// TwinCAT 3 PLC project AstroBROT
// Title: AstroBROT
// Company: BROT
// ProjectVersion: 0.4.5
// ProgramVersion: 3.1.4026.11
// libraries:
//   Tc2_Math, * (Beckhoff Automation GmbH)
//   Tc2_Standard, * (Beckhoff Automation GmbH)
//   Tc2_System, * (Beckhoff Automation GmbH)
//   Tc2_Utilities, * (Beckhoff Automation GmbH)
//   Tc3_Module, * (Beckhoff Automation GmbH)
// project tree:
//   POUs/FUNCTIONS/ ATAN2.TcPOU, CO_REFRACT_FORWARD.TcPOU, CT2LST.TcPOU, DateTime2JD.TcPOU, JD2LST.TcPOU, JD2JEPOCH.TcPOU, JD2OBLIQUITY.TcPOU, LMST2LAST.TcPOU, TEN.TcPOU
//   POUs/FUNCTION_BLOCKS/ FB_ALTAZ2HADEC.TcPOU, FB_CO_ABERRATION.TcPOU, FB_CO_REFRACT.TcPOU, FB_CO_NUTATE.TcPOU, FB_EQ2HOR.TcPOU, FB_HADEC2RADEC.TcPOU, FB_HADEC2ALTAZ.TcPOU, FB_HOR2EQ.TcPOU, FB_IAU2000B.TcPOU, FB_PRECESS.TcPOU, FB_RADEC2HADEC.TcPOU, FB_SUNPOS.TcPOU
//   GVLs/ Global_Version.TcGVL

// ---- GVLs/Global_Version.TcGVL
{attribute 'qualified_only'}
VAR_GLOBAL CONSTANT
	// Mirrors Beckhoff's own Global_Version.stLibVersion_* pattern (see ST_LibVersion),
	// which only covers Tc2_*/Tc3_* library references, not custom ones -- until now: this
	// GVL uses Beckhoff's own naming exactly, so it merges into a consumer's Global_Version.
	// Kept in sync with <ProjectVersion> in AstroBROT.plcproj at release time.
	stLibVersion_AstroBROT : ST_LibVersion := (
		iMajor := 0,
		iMinor := 4,
		iBuild := 5,
		iRevision := 0,
		nFlags := 1,
		sVersion := '0.4.5'
	);
END_VAR

// ---- POUs/FUNCTIONS/ATAN2.TcPOU
FUNCTION ATAN2 : LREAL
VAR_INPUT
	y		: LREAL;
	x		: LREAL;
END_VAR
VAR
END_VAR

(* source: https://de.wikipedia.org/wiki/Arctan2 *)
ATAN2 := 0.0;

IF x > 0 THEN
	ATAN2 := ATAN(y/x);
ELSIF x < 0 AND y > 0 THEN
	ATAN2 := ATAN(y/x) + PI;
ELSIF x < 0 AND y = 0 THEN
	ATAN2 := PI;
ELSIF x < 0 AND y < 0 THEN
	ATAN2 := ATAN(y/x) - PI;
ELSIF x = 0 AND y > 0 THEN
	ATAN2 := PI/2.0;
ELSIF x = 0 AND y < 0 THEN
	ATAN2 := -PI/2.0;
END_IF

END_FUNCTION

// ---- POUs/FUNCTIONS/CO_REFRACT_FORWARD.TcPOU
FUNCTION CO_REFRACT_FORWARD : LREAL
VAR_INPUT
	a			: LREAL; 			// The observed (apparent) altitude, in DEGREES.
	P			: LREAL := 1010.0;	// Pressure [in millibars]. Default is 1010 millibars.
	T			: LREAL := 0.0;		// Ground Temp [in Celsius].  Default is 0 Celsius.
END_VAR
VAR_OUTPUT
	clamped		: BOOL;				// TRUE if a, P or T was outside its valid range and has been limited
END_VAR
VAR
	ref			: LREAL;
	ref_lo		: LREAL;
	ref_hi		: LREAL;
	w			: LREAL;
	tk, gamma, beta, tan_z	: LREAL;
END_VAR
VAR CONSTANT
	d2r 		: LREAL := PI/180.0;
	// (n-1) * T / P for dry air at 0.55 um (IAG 1999 optical refractivity, as in eraRefco)
	k_gamma		: LREAL := 7.902649953145277E-5;
	// The two branches are blended linearly between these altitudes [DEGREES], so there is no step
	a_blend_lo	: LREAL := 14.0;
	a_blend_hi	: LREAL := 16.0;
END_VAR

(*Atmospheric refraction in DEGREES for an OBSERVED altitude a, pressure P [mbar] and temperature T [degC].
Dry air, 0.55 um, no humidity or wavelength input.

Below a_blend_lo (about 14 deg): the rational formula of the Explanatory Supplement to the Astronomical
Almanac, 2013, p.280 (eq. 7.91, not checked against the book).
From a_blend_hi (about 16 deg): dZ = A tan Z + B tan^3 Z with A and B from Green, Spherical Astronomy, 1987,
eq. 4.31 and beta from Stone (1996), exactly as ERFA's eraRefco (dry, wl = 0.55 um). eraRefco is
Copyright (C) 2013-2023 NumFOCUS Foundation, derived from SOFA, see NOTICE-erfa.md. Its documentation gives
62 mas worst case against ray tracing for zenith distances 15 to 75 deg (optical, humid air included).
Between the two: linear blend, so the result is continuous.

Accuracy of this implementation against an independent ray trace (testing/check_refraction_model.py, P 900 to
1013 mbar, T -15 to 30 degC): within 0.7 arcsec from 15 deg up, within 1.9 arcsec from 10 to 15 deg. NOT verified
below 10 deg, where the error reaches about 6 arcsec at 5 deg; do not rely on it near the horizon.

a, P and T are limited to [0, 90], [600, 1200] and [-40, 40] and clamped is set, so a caller can tell. A
below-horizon altitude therefore gets the horizon refraction.*)

clamped := (a < 0.0) OR (a > 90.0) OR (P < 600.0) OR (P > 1200.0) OR (T < -40.0) OR (T > 40.0);
a := LIMIT(0.0, a, 90.0);
P := LIMIT(600.0, P, 1200.0);
T := LIMIT(-40.0, T, 40.0);

IF a < a_blend_hi THEN
	ref_lo := P/(T+273.0)* (0.1594 + 0.0196 * a + 0.00002 * EXPT(a, 2)) / (1.0 + 0.505 * a + 0.0845 * EXPT(a, 2));
END_IF

IF a > a_blend_lo THEN
	tk := T + 273.15;
	gamma := k_gamma * P / tk;
	beta := 4.4474E-6 * tk;
	tan_z := TAN((90.0 - a) * d2r);
	ref_hi := (gamma * (1.0 - beta) * tan_z - gamma * (beta - gamma / 2.0) * tan_z * tan_z * tan_z) / d2r;
END_IF

IF a <= a_blend_lo THEN
	ref := ref_lo;
ELSIF a >= a_blend_hi THEN
	ref := ref_hi;
ELSE
	w := (a - a_blend_lo) / (a_blend_hi - a_blend_lo);
	ref := (1.0 - w) * ref_lo + w * ref_hi;
END_IF
CO_REFRACT_FORWARD :=  ref;

END_FUNCTION

// ---- POUs/FUNCTIONS/CT2LST.TcPOU
FUNCTION CT2LST : LREAL
VAR_INPUT
	lng: LREAL; // The longitude in degrees (east of Greenwich) of the place for which the local sidereal time is desired, scalar.   The Greenwich mean sidereal time (GMST) can be found by setting Lng = 0.
	jd:	LREAL; // this is the Julian date of time in question
END_VAR
VAR
	t0,t,theta: LREAL;
END_VAR
VAR CONSTANT
	jd2000: LREAL := 2451545.0;
END_VAR

(* https://github.com/wlandsman/IDLAstro/blob/master/pro/ct2lst.pro 

;+
; NAME:
;     CT2LST
; PURPOSE:
;     To convert from Local Civil Time to Local Mean Sidereal Time.
;
; CALLING SEQUENCE:
;     CT2LST, Lst, Lng, Tz, Time, [Day, Mon, Year] 
;                       or
;     CT2LST, Lst, Lng, dummy, JD
;
; INPUTS:
;     Lng  - The longitude in degrees (east of Greenwich) of the place for 
;            which the local sidereal time is desired, scalar.   The Greenwich 
;            mean sidereal time (GMST) can be found by setting Lng = 0.
;     Tz  - The time zone of the site in hours, positive East  of the Greenwich
;           meridian (ahead of GMT).  Use this parameter to easily account 
;           for Daylight Savings time (e.g. -4=EDT, -5 = EST/CDT), scalar
;           This parameter is not needed (and ignored) if Julian date is 
;           supplied.    ***Note that the sign of TZ was changed in July 2008
;           to match the standard definition.*** 
;     Time or JD  - If more than four parameters are specified, then this is 
;               the time of day of the specified date in decimal hours.  If 
;               exactly four parameters are specified, then this is the 
;               Julian date of time in question, scalar or vector
;
; OPTIONAL INPUTS:
;      Day -  The day of the month (1-31),integer scalar or vector
;      Mon -  The month, in numerical format (1-12), integer scalar or vector
;      Year - The 4 digit year (e.g. 2008), integer scalar or vector
;
; OUTPUTS:
;       Lst   The Local Sidereal Time for the date/time specified in hours.
;
; RESTRICTIONS:
;       If specified, the date should be in numerical form.  The year should
;       appear as yyyy.
;
; PROCEDURE:
;       The Julian date of the day and time is question is used to determine
;       the number of days to have passed since 0 Jan 2000.  This is used
;       in conjunction with the GST of that date to extrapolate to the current
;       GST; this is then used to get the LST.    See Astronomical Algorithms
;       by Jean Meeus, p. 84 (Eq. 11-4) for the constants used.
;
; EXAMPLE:
;       Find the Greenwich mean sidereal time (GMST) on 2008 Jul 30 at 15:53 pm
;       in Baltimore, Maryland (longitude=-76.72 degrees).   The timezone is 
;       EDT or tz=-4
;
;       IDL> CT2LST, lst, -76.72, -4,ten(15,53), 30, 07, 2008
;
;               ==> lst =  11.356505  hours  (= 11h 21m 23.418s)
;
;       The Web site  http://tycho.usno.navy.mil/sidereal.html contains more
;       info on sidereal time, as well as an interactive calculator.
; PROCEDURES USED:
;       jdcnv - Convert from year, month, day, hour to julian date
;
; MODIFICATION HISTORY:
;     Adapted from the FORTRAN program GETSD by Michael R. Greason, STX, 
;               27 October 1988.
;     Use IAU 1984 constants Wayne Landsman, HSTX, April 1995, results 
;               differ by about 0.1 seconds  
;     Longitudes measured *east* of Greenwich   W. Landsman    December 1998
;     Time zone now measure positive East of Greenwich W. Landsman July 2008
;     Remove debugging print statement  W. Landsman April 2009
;-

*)

t0 := jd - jd2000;
t := t0/36525.0;
// Compute GST in seconds.
theta := 280.46061837 + (360.98564736629 * t0) + EXPT(t, 2)*(0.000387933 - (t/ 3871.0E4));
//theta := 100.46061837 + 36000.770053608*t0 + 0.000387933*EXPT(t0,2) - EXPT(t0,3)/3871000.0;
// Compute LST in hours.
CT2LST := ( theta + lng)/15.0;
CT2LST := MODABS(CT2LST, 24.0);

END_FUNCTION

// ---- POUs/FUNCTIONS/DateTime2JD.TcPOU
FUNCTION DateTime2JD : LREAL
VAR_INPUT
	epoch			: TIMESTRUCT;
END_VAR
VAR
	a, y, m, jdn	: LREAL;
END_VAR

// Julian Date of a TIMESTRUCT (Meeus, Astronomical Algorithms, ch. 7; integer-day formula of the Gregorian calendar).
//
// - epoch must be UTC. The function does not convert or check the time zone; a local time gives a JD that is off by the
//   UTC offset, and with it the sidereal time (15 degrees per hour).
// - Gregorian calendar only, i.e. valid from 1582-10-15. Earlier dates would need the Julian-calendar formula.
// - No validation. Out-of-range fields roll over (month 13 is January of the next year, 30 February is 2 March), and an
//   all-zero TIMESTRUCT (e.g. a clock that has not been synchronised yet) gives 1721027.5, which is not a usable time.
a := FLOOR((14.0 - epoch.wMonth)/12.0);
y := epoch.wYear + 4800.0 - a;
m := epoch.wMonth + 12.0*a - 3.0;

jdn := epoch.wDay + FLOOR((153*m + 2)/5) + 365.0*y + FLOOR(y/4) - FLOOR(y/100) + FLOOR(y/400) - 32045.0;

DateTime2JD := jdn
			+ (epoch.wHour-12.0)/24.0
			+ (epoch.wMinute/1440.0) 
			+ (epoch.wSecond/86400.0)
			+ (DWORD_TO_REAL(epoch.wMilliseconds)/86400000.0);

END_FUNCTION

// ---- POUs/FUNCTIONS/JD2LST.TcPOU
FUNCTION JD2LST : LREAL
VAR_INPUT
	jd			: LREAL;	// Julian date, UTC time scale
	lon			: LREAL;	// longitude in degrees
	dut1		: LREAL := 0.0;	// UT1-UTC in seconds (IERS, |dut1| < 0.9), 0 treats UTC as UT1
END_VAR
VAR
	ut1			: LREAL;
	T			: LREAL;
	theta0		: LREAL;
END_VAR
VAR CONSTANT
	jd2000		: LREAL := 2451545.0;
END_VAR

// following https://squarewidget.com/astronomical-calculations-sidereal-time/
ut1 := jd + dut1 / 86400.0;
T := ((ut1 - jd2000) / 36525.0);
theta0 := 280.46061837 + 360.98564736629 * (ut1 - jd2000) + (0.000387933 * T * T) - (T * T * T / 38710000.0); // (12.4)

// LST is only defined from 0 to 360
JD2LST := MODABS(theta0 + lon, 360.0); // LST in degrees

END_FUNCTION

// ---- POUs/FUNCTIONS/JD2JEPOCH.TcPOU
FUNCTION JD2JEPOCH : LREAL
VAR_INPUT
	jd			: LREAL;	// Julian date
END_VAR
VAR CONSTANT
	jd2000		: LREAL := 2451545.0;
END_VAR

// Julian epoch (equinox) of jd, e.g. for precession
JD2JEPOCH := (jd - jd2000)/365.25 + 2000.0;

END_FUNCTION

// ---- POUs/FUNCTIONS/JD2OBLIQUITY.TcPOU
FUNCTION JD2OBLIQUITY : LREAL
VAR_INPUT
	jd			: LREAL;	// Julian date
	d_eps		: LREAL;	// nutation in obliquity in arcsec (FB_IAU2000B)
END_VAR
VAR
	T			: LREAL;
	eps0		: LREAL;
END_VAR
VAR CONSTANT
	d2r			: LREAL := PI/180.0;
	jd2000		: LREAL := 2451545.0;
END_VAR

// Julian centuries from J2000 of jd
T := (jd - jd2000)/36525.0;

// mean obliquity of the ecliptic in arcsec
eps0 := 23.4392911*3600.0 - 46.8150*T - 0.00059*EXPT(T, 2) + 0.001813*EXPT(T, 3);

// TRUE obliquity of the ecliptic in radians
JD2OBLIQUITY := (eps0 + d_eps)/3600.0*d2r;

END_FUNCTION

// ---- POUs/FUNCTIONS/LMST2LAST.TcPOU
FUNCTION LMST2LAST : LREAL
VAR_INPUT
	lmst		: LREAL;	// local mean sidereal time in degrees
	d_psi		: LREAL;	// nutation in longitude in arcsec (FB_IAU2000B)
	eps			: LREAL;	// TRUE obliquity of the ecliptic in radians (JD2OBLIQUITY)
END_VAR

// local APPARENT sidereal time in degrees: add the equation of the equinoxes
LMST2LAST := lmst + d_psi*COS(eps)/3600.0;

END_FUNCTION

// ---- POUs/FUNCTIONS/TEN.TcPOU
FUNCTION TEN : LREAL
VAR_INPUT
	dd, mm, ss	: LREAL;
END_VAR
VAR
	fSign	: LREAL;
END_VAR

// as IDLAstro's ten: a minus sign on any element makes the whole value negative, so TEN(-5, 30, 0) = -5.5
// (unlike IDL, a literal -0.0 is not recognised as negative)
IF (dd < 0.0) OR (mm < 0.0) OR (ss < 0.0) THEN
	fSign := -1.0;
ELSE
	fSign := 1.0;
END_IF
TEN := fSign * (ABS(dd) + (ABS(mm)/60.0) + (ABS(ss)/3600.0));

END_FUNCTION

// ---- POUs/FUNCTION_BLOCKS/FB_ALTAZ2HADEC.TcPOU
FUNCTION_BLOCK FB_ALTAZ2HADEC
VAR_INPUT
	alt			: LREAL;	// the local apparent altitude, in DEGREES
	az			: LREAL;	// the local apparent azimuth, in DEGREES
	lat			: LREAL;	// the local geodetic latitude, in DEGREES
END_VAR
VAR_OUTPUT
	ha			: LREAL;	// the local apparent hour angle, in DEGREES
	dec			: LREAL;	// the local apparent declination, in DEGREES
END_VAR
VAR
	alt_r		: LREAL;
	az_r		: LREAL;
	lat_r		: LREAL;
	sindec		: LREAL;
END_VAR
VAR CONSTANT
	d2r			: LREAL := PI/180.0;
	r2d			: LREAL := 180.0/PI;
	//h2r:	LREAL := PI/12.0;
	//h2d:	LREAL := 15.0;
END_VAR

(*https://github.com/wlandsman/IDLAstro/blob/master/pro/

  NAME:
    ALTAZ2HADEC
 PURPOSE:
    Convert Horizon (Alt-Az) coordinates to Hour Angle and Declination.
 EXPLANATION::
    Can deal with the NCP singularity.    Intended mainly to be used by
    program hor2eq.pro
 CALLING SEQUENCE:
   ALTAZ2HADEC, alt, az, lat, ha, dec

 INPUTS
   alt - the local apparent altitude, in DEGREES, scalar or vector
   az  - the local apparent azimuth, in DEGREES, scalar or vector,
         measured EAST of NORTH!!!  If you have measured azimuth west-of-south
        (like the book MEEUS does), convert it to east of north via:
                       az = (az + 180) mod 360

   lat -  the local geodetic latitude, in DEGREES, scalar or vector.

 OUTPUTS
   ha  -  the local apparent hour angle, in DEGREES.  The hour angle is the 
          time that right ascension of 0 hours crosses the local meridian.  
          It is unambiguously defined.
   dec -  the local apparent declination, in DEGREES.

 EXAMPLE:
     Arcturus is observed at an apparent altitude of 59d,05m,10s and an 
     azimuth (measured east of north) of 133d,18m,29s while at the 
     latitude of +43.07833 degrees.
     What are the local hour angle and declination of this object?

     IDL> altaz2hadec, ten(59,05,10), ten(133,18,29), 43.07833, ha, dec
     ===> Hour angle ha = 336.683 degrees
          Declination, dec = 19.1824 degrees

       The widely available XEPHEM code gets:
                 Hour Angle = 336.683
                 Declination = 19.1824

 REVISION HISTORY:
    Written  Chris O'Dell Univ. of Wisconsin-Madison May 2002*)

alt_r  := alt*d2r;
az_r := az*d2r;
lat_r := lat*d2r;

//******************************************************************************
// find local HOUR ANGLE (in degrees, from 0. to 360.)
ha := atan2( (-SIN(az_r)*COS(alt_r)), (-COS(az_r)*SIN(lat_r)*COS(alt_r)+SIN(alt_r)*COS(lat_r)));
ha := ha / d2r;
IF ha < 0.0 THEN 
	ha := ha + 360.0;
END_IF
ha := MODABS(ha, 360.0);

// Find declination (positive if north of Celestial Equator, negative if south)
sindec := SIN(lat_r)*SIN(alt_r) + COS(lat_r)*COS(alt_r)*COS(az_r);
// convert dec to degrees
dec := ASIN(LIMIT(-1.0, sindec, 1.0))/d2r;   // clamp: at the celestial pole rounding gives 1 + 2.2E-16, and ASIN of that is NaN

END_FUNCTION_BLOCK

// ---- POUs/FUNCTION_BLOCKS/FB_CO_ABERRATION.TcPOU
FUNCTION_BLOCK FB_CO_ABERRATION
VAR_INPUT
	jd			: LREAL;		// Julian Date
	ra			: LREAL;		// RA in degrees
	dec			: LREAL; 		// Dec in degrees
	eps 		: LREAL := 0.0;
END_VAR
VAR_OUTPUT
	d_ra		: LREAL;
	d_dec		: LREAL;
END_VAR
VAR
	sunpos		: FB_SUNPOS;
	nutate		: FB_IAU2000B;
	sunra		: LREAL;
	sundec		: LREAL;
	sunlon		: LREAL;
	d_psi		: LREAL;
	d_epsilon	: LREAL; 
	eps_loc		: LREAL;		// obliquity in radians, eps or calculated if eps = 0
	t, e, peri, cd, sd, ce, te, cp, sp, cs, ss, ca, sa, term1, term2, term3, term4: LREAL;
END_VAR
VAR CONSTANT
	d2r 		: LREAL := PI/180.0;
	k			: LREAL := 20.49552; 	//constant of aberration, in arcseconds
	
END_VAR

(* https://github.com/wlandsman/IDLAstro/blob/master/pro/co_aberration.pro
;+
;  NAME:
;     CO_ABERRATION
; PURPOSE:
;     Calculate changes to Ra and Dec due to the effect of annual aberration 
; EXPLANATION:
;      as described in Meeus, Chap 23.
; CALLING SEQUENCE:
;      co_aberration, jd, ra, dec, d_ra, d_dec, [EPS = ]
; INPUTS
;       jd      : Julian Date [scalar or vector]
;       ra, dec : ra  and dec's in degrees
;
; OUTPUTS
;       d_ra, d_dec: the corrections to ra and dec due to aberration in 
;                    degrees.  (These values can be added to the true RA 
;                    and dec to get the apparent position).   Note that d_ra
;                     is *not* multiplied by cos(dec), so that 
;                     apparent_ra = ra + d_ra. 
; OPTIONAL INPUT KEYWORD:
;       eps : set this to the true obliquity of the ecliptic (in radians), or
;         it will be set for you if you don't know it (in that case, set it to
;                 an empty variable).
; NOTES:
;  These formula are from Meeus, Chapters 23.  Accuracy is much better than 1 
;   arcsecond.
;
;   The maximum deviation due to annual aberration is 20.49" and occurs when the
;   Earth velocity is perpendicular to the direction of the star.
;
; REVISION HISTORY:
;   Written, June 2002,      Chris O'Dell, U. of Wisconsin
;   Fix error with vector input   W. Landsman   June 2009
;   June 2009 update fixed case where JD was scalar but RA,Dec were vectors, but 
;     broke the case when both JD and RA,Dec were vectors Aug 2012 W. Landsman
;   Further fix when JD is 1 element vector  W. Landsman
;
;	UPDATE: HAS BEEN REWORKED FOR THE COORD STRUCTURE -> OUTPUT IS IN DEGREES
*)

T := (jd -2451545.0)/36525.0; // julian centuries from J2000 of jd.

IF eps = 0.0 THEN
	// must calculate obliquity of ecliptic
	nutate(jd := jd,
		d_psi => d_psi, 
		d_eps => d_epsilon); //d_psi and d_epsilon in arcsec
	// TRUE obliquity OF the ecliptic in radians
	eps_loc := JD2OBLIQUITY(jd, d_epsilon);
ELSE
	eps_loc := eps;
END_IF

sunpos(jd := jd, ra => sunra, dec => sundec, longmed => sunlon);

// Earth's orbital eccentricity
e := 0.016708634 - 0.000042037*T - 0.0000001267*EXPT(T, 2);
// longitude of perihelion, in degrees 
peri := 102.93735 + 1.71946*T + 0.00046*EXPT(T, 2);

//Useful Trig Functions
cd := COS(dec*d2r);		sd := SIN(dec*d2r);
ce := COS(eps_loc); 	te := TAN(eps_loc);
cp := COS(peri*d2r);	sp := SIN(peri*d2r);
cs := COS(sunlon*d2r);	ss := SIN(sunlon*d2r);
ca := COS(ra*d2r);		sa := SIN(ra*d2r);

term1 := (ca*cs*ce + sa*ss)/cd;
term2 := (ca*cp*ce + sa*sp)/cd;
term3 := (cs*ce*(te*cd - sa*sd) + ca*sd*ss);
term4 := (cp*ce*(te*cd - sa*sd) + ca*sd*sp);

d_ra := (-k * term1 + e*k * term2)/3600;
d_dec := (-k * term3 + e*k * term4)/3600;

END_FUNCTION_BLOCK

// ---- POUs/FUNCTION_BLOCKS/FB_SUNPOS.TcPOU
FUNCTION_BLOCK FB_SUNPOS
VAR_INPUT
	jd				: LREAL;		// Julian Date
END_VAR
VAR_OUTPUT
	ra				: LREAL;		// right ascension
	dec				: LREAL;		// declination of the sun 
	longmed			: LREAL;		// longitude
	oblt			: LREAL;		// True Obliquity
END_VAR
VAR
	t				: LREAL;		//  Julian centuries FROM 1900.0
	l				: LREAL;		//  sun's mean longitude
	me				: LREAL;		// Earth's mean anomaly
	ellcor			: LREAL;		// ellipticity of the orbit
	mv				: LREAL;		// mean anomaly of Venus
	vencorr			: LREAL;		
	mm				: LREAL;		
	marscorr		: LREAL;		
	mj				: LREAL;		
	jupcorr			: LREAL;		
	d				: LREAL;		
	longterm		: LREAL;		
	mooncorr		: LREAL;		
	omega			: LREAL;
END_VAR
VAR CONSTANT
	d2r				: LREAL := PI/180.0; // Pi/180
END_VAR

(* https://github.com/wlandsman/IDLAstro/blob/master/pro/
NOTES:
;       Patrick Wallace (Rutherford Appleton Laboratory, UK) has tested the
;       accuracy of a C adaptation of the sunpos.pro code and found the 
;       following results.   From 1900-2100 SUNPOS  gave 7.3 arcsec maximum 
;       error, 2.6 arcsec RMS.  Over the shorter interval 1950-2050 the figures
;       were 6.4 arcsec max, 2.2 arcsec RMS.  
;
;       The returned ra and Dec are in the given date's equinox.
;
;       Procedure was extensively revised in May 1996, and the new calling
;       sequence is incompatible with the old one.source: https://idlastro.gsfc.nasa.gov/ftp/pro/astro/sunpos.pro *)

//  form TIME in Julian centuries FROM 1900.0
t := (jd - 2415020.0) / 36525.0;

//  form sun's mean longitude
l := (279.696678 + LMOD(36000.768925 * t, 360.0)) * 3600.0;

//  allow for ellipticity of the orbit (equation of centre) using the Earth's mean anomaly ME
me := 358.475844 + LMOD(35999.049750 * t, 360.0);
ellcor  := (6910.1 - 17.2 * t) * SIN(me * d2r) + 72.3 * SIN(2.0 * me*d2r);
l := l + ellcor;
 
// allow FOR the Venus perturbations using the mean anomaly OF Venus MV
mv := 212.603219 + LMOD(58517.803875 * t, 360.0);
vencorr := 4.8 * COS((299.1017 + mv - me)*d2r) + 
           5.5 * COS((148.3133 +  2.0 * mv  -  2.0 * me )*d2r) + 
           2.5 * COS((315.9433 +  2.0 * mv  -  3.0 * me )*d2r) + 
           1.6 * COS((345.2533 +  3.0 * mv  -  4.0 * me )*d2r) + 
           1.0 * COS((318.15   +  3.0 * mv  -  5.0 * me )*d2r);
l := l + vencorr;

//  Allow FOR the Mars perturbations using the mean anomaly OF Mars MM
mm := 319.529425  +  LMOD( 19139.858500 * t,  360.0 );
marscorr := 2.0 * COS((343.8883 -  2.0 * mm  +  2.0 * me)*d2r ) + 
            1.8 * COS((200.4017 -  2.0 * mm  + me) * d2r);
l := l + marscorr;

// Allow FOR the Jupiter perturbations using the mean anomaly OF Jupiter MJ
mj := 225.328328  +  LMOD( 3034.6920239 * t,  360.0 );
jupcorr := 7.2 * COS(( 179.5317 - mj + me )*d2r) + 
           2.6 * COS((263.2167  -  MJ ) *d2r) + 
           2.7 * COS(( 87.1450  -  2.0 * mj  +  2.0 * me ) *d2r) + 
           1.6 * COS((109.4933  -  2.0 * mj  +  me ) *d2r);
l := l + jupcorr;

// Allow FOR the Moons perturbations using the mean elongation OF the Moon from the Sun D
d := 350.7376814  + LMOD(445267.11422 * t,  360.0);
mooncorr  := 6.5 * SIN(d * d2r);
l := l + mooncorr;

// Allow for long period terms
longterm := 6.4 * SIN((231.19  +  20.20 * t) * d2r);
l :=  l + longterm;
l :=  LMOD(l + 2592000.0,  1296000.0); 
longmed := l / 3600.0;

// Allow for Aberration
l :=  l - 20.5;

// Allow for Nutation using the longitude of the Moons mean node OMEGA
omega := 259.183275 - LMOD(1934.142008 * t, 360.0);
l :=  l - 17.2 * SIN(omega * d2r);

// Form the True Obliquity
oblt := 23.452294 - 0.0130125 * t + (9.2 * COS(omega * d2r)) / 3600.0;

// Form Right Ascension AND Declination
l := l / 3600.0;
ra := ATAN2(SIN(l * d2r) * COS(oblt * d2r), COS(l * d2r));
dec := ASIN(SIN(l * d2r) * SIN(oblt * d2r));
 
ra := ra/d2r;
ra := MODABS(ra, 360.0);
dec := dec/d2r;

END_FUNCTION_BLOCK

// ---- POUs/FUNCTION_BLOCKS/FB_IAU2000B.TcPOU
FUNCTION_BLOCK FB_IAU2000B
VAR_INPUT
	jd: LREAL;
END_VAR
VAR_OUTPUT
	// unit: arcsec
	// d_psi and d_eps are not the pure IAU 2000B nutation: constant offsets standing in for the planetary terms
	// and the frame bias are added (-0.0433585 and -0.0084531 arcsec, see the end of the implementation)
	d_psi : LREAL := 0.0; 
	d_eps : LREAL := 0.0;
END_VAR
VAR
	t	: LREAL;
	m_l, m_l_, m_f, m_d, m_om : LREAL;
	theta, s_theta, c_theta : LREAL;
	d_p, d_e : LREAL := 0.0;
	i : INT;
END_VAR
VAR CONSTANT
	d2r				: LREAL := PI/180.0;
	asec2r			: LREAL := PI/(180*3600);
	asec360			: LREAL := 3600*360;
	jd2000			: LREAL := 2451545.0;
	// number of luni-solar terms of IAU 2000B
	n_terms			: INT := 77;
	// Luni-Solar argument multipliers:
	l	: ARRAY[1..77] OF LREAL := [0, 0, 0, 0, 0, 0, 1, 0, 1, 0, 0, -1, -1, 1, -1, -1, 1, -2, 0, 0, 0, -2, 2, 1, -1, 2, 0, 0, -1, 0, 0, 1, 0, -1, 0, 1, -2, 0, 0, 0, 0, 1, 2, -2, 2, 0, 0, -1, 2, 1, 0, 1, -2, 3, 0, 1, 0, -1, -1, 0, -2, 1, 2, -1, 1, 1, -1, 1, -1, 0, -1, -1, 0, 1, -2, -1, 1];
	l_	: ARRAY[1..77] OF LREAL := [0, 0, 0, 0, 1, 1, 0, 0, 0, -1, 0, 0, 0, 0, 0, 0, 0, 0, 0, 0, -2, 0, 0, 0, 0, 0, 0, 1, 0, 2, 0, 0, -1, 0, 2, 0, 0, 1, 0, -1, 0, 0, 0, 0, 0, -1, 0, -1, 0, 0, 1, -1, 0, 0, -1, -1, 0, -1, 0, -1, 0, 1, 0, 1, 1, 0, 0, 0, 0, 0, 0, 1, -2, 0, 0, 0, 1];
	f 	: ARRAY[1..77] OF LREAL := [0, 2, 2, 0, 0, 2, 0, 2, 2, 2, 2, 2, 0, 0, 0, 2, 2, 2, 0, 2, 2, 0, 2, 2, 2, 0, 2, 0, 0, 2, -2, 0, 0, 2, 0, 2, 2, 2, 2, 2, 0, 2, 2, 0, 2, 2, 0, 0, 0, 0, 2, 0, 2, 2, 0, 2, 0, 2, 2, 2, 0, 2, 0, 0, 0, 2, 2, 0, 0, 2, 2, 0, 2, 2, 2, 0, 2];
	d 	: ARRAY[1..77] OF LREAL := [0, -2, 0, 0, 0, -2, 0, 0, 0, -2, -2, 0, 2, 0, 0, 2, 0, 0, 2, 2, -2, 2, 0, -2, 0, 0, 0, 0, 2, -2, 2, -2, 0, 2, 0, 2, 0, 0, 2, 0, 2, -2, -2, 2, 0, -2, -2, 2, -2, 2, -2, 0, 0, 0, 2, 0, 1, 2, 0, 2, 0, 0, 0, 1, 0, 0, -2, 0, 1, 1, 4, 1, -2, 2, 2, 0, -2];
	om	: ARRAY[1..77] OF LREAL := [1, 2, 2, 2, 0, 2, 0, 1, 2, 2, 1, 2, 0, 1, 1, 2, 1, 1, 0, 2, 2, 0, 2, 2, 1, 0, 0, 1, 1, 2, 0, 1, 1, 1, 0, 2, 0, 2, 1, 2, 1, 1, 2, 1, 1, 1, 1, 0, 1, 0, 1, 0, 2, 2, 0, 2, 0, 2, 0, 2, 1, 2, 1, 0, 0, 0, 1, 2, 0, 2, 2, 1, 1, 1, 2, 2, 2];
	//  Luni-Solar nutation coefficients, unit 1e-7 arcsec:
	A 	: ARRAY[1..77] OF LREAL := [-172064161.0, -13170906.0, -2276413.0, 2074554.0, 1475877.0, -516821.0, 711159.0, -387298.0, -301461.0, 215829.0, 128227.0, 123457.0, 156994.0, 63110.0, -57976.0, -59641.0, -51613.0, 45893.0, 63384.0, -38571.0, 32481.0, -47722.0, -31046.0, 28593.0, 20441.0, 29243.0, 25887.0, -14053.0, 15164.0, -15794.0, 21783.0, -12873.0, -12654.0, -10204.0, 16707.0, -7691.0, -11024.0, 7566.0, -6637.0, -7141.0, -6302.0, 5800.0, 6443.0, -5774.0, -5350.0, -4752.0, -4940.0, 7350.0, 4065.0, 6579.0, 3579.0, 4725.0, -3075.0, -2904.0, 4348.0, -2878.0, -4230.0, -2819.0, -4056.0, -2647.0, -2294.0, 2481.0, 2179.0, 3276.0, -3389.0, 3339.0, -1987.0, -1981.0, 4026.0, 1660.0, -1521.0, 1314.0, -1283.0, -1331.0, 1383.0, 1405.0, 1290.0];
	A1 	: ARRAY[1..77] OF LREAL := [-174666.0, -1675.0, -234.0, 207.0, -3633.0, 1226.0, 73.0, -367.0, -36.0, -494.0, 137.0, 11.0, 10.0, 63.0, -63.0, -11.0, -42.0, 50.0, 11.0, -1.0, 0.0, 0.0, -1.0, 0.0, 21.0, 0.0, 0.0, -25.0, 10.0, 72.0, 0.0, -10.0, 11.0, 0.0, -85.0, 0.0, 0.0, -21.0, -11.0, 21.0, -11.0, 10.0, 0.0, -11.0, 0.0, -11.0, -11.0, 0.0, 0.0, 0.0, 0.0, 0.0, 0.0, 0.0, 0.0, 0.0, 0.0, 0.0, 0.0, 0.0, 0.0, 0.0, 0.0, 0.0, 0.0, 0.0, 0.0, 0.0, 0.0, 0.0, 0.0, 0.0, 0.0, 0.0, 0.0, 0.0, 0.0];
	A2 	: ARRAY[1..77] OF LREAL := [33386.0, -13696.0, 2796.0, -698.0, 11817.0, -524.0, -872.0, 380.0, 816.0, 111.0, 181.0, 19.0, -168.0, 27.0, -189.0, 149.0, 129.0, 31.0, -150.0, 158.0, 0.0, -18.0, 131.0, -1.0, 10.0, -74.0, -66.0, 79.0, 11.0, -16.0, 13.0, -37.0, 63.0, 25.0, -10.0, 44.0, -14.0, -11.0, 25.0, 8.0, 2.0, 2.0, -7.0, -15.0, 21.0, -3.0, -21.0, -8.0, 6.0, -24.0, 5.0, -6.0, -2.0, 15.0, -10.0, 8.0, 5.0, 7.0, 5.0, 11.0, -10.0, -7.0, -2.0, 1.0, 5.0, -13.0, -6.0, 0.0, -353.0, -5.0, 9.0, 0.0, 0.0, 8.0, -2.0, 4.0, 0.0];
	B 	: ARRAY[1..77] OF LREAL := [92052331.0, 5730336.0, 978459.0, -897492.0, 73871.0, 224386.0, -6750.0, 200728.0, 129025.0, -95929.0, -68982.0, -53311.0, -1235.0, -33228.0, 31429.0, 25543.0, 26366.0, -24236.0, -1220.0, 16452.0, -13870.0, 477.0, 13238.0, -12338.0, -10758.0, -609.0, -550.0, 8551.0, -8001.0, 6850.0, -167.0, 6953.0, 6415.0, 5222.0, 168.0, 3268.0, 104.0, -3250.0, 3353.0, 3070.0, 3272.0, -3045.0, -2768.0, 3041.0, 2695.0, 2719.0, 2720.0, -51.0, -2206.0, -199.0, -1900.0, -41.0, 1313.0, 1233.0, -81.0, 1232.0, -20.0, 1207.0, 40.0, 1129.0, 1266.0, -1062.0, -1129.0, -9.0, 35.0, -107.0, 1073.0, 854.0, -553.0, -710.0, 647.0, -700.0, 672.0, 663.0, -594.0, -610.0, -556.0];
	B1 	: ARRAY[1..77] OF LREAL := [9086.0, -3015.0, -485.0, 470.0, -184.0, -677.0, 0.0, 18.0, -63.0, 299.0, -9.0, 32.0, 0.0, 0.0, 0.0, -11.0, 0.0, -10.0, 0.0, -11.0, 0.0, 0.0, -11.0, 10.0, 0.0, 0.0, 0.0, -2.0, 0.0, -42.0, 0.0, 0.0, 0.0, 0.0, -1.0, 0.0, 0.0, 0.0, 0.0, 0.0, 0.0, 0.0, 0.0, 0.0, 0.0, 0.0, 0.0, 0.0, 0.0, 0.0, 0.0, 0.0, 0.0, 0.0, 0.0, 0.0, 0.0, 0.0, 0.0, 0.0, 0.0, 0.0, 0.0, 0.0, 0.0, 0.0, 0.0, 0.0, 0.0, 0.0, 0.0, 0.0, 0.0, 0.0, 0.0, 0.0, 0.0];
	B2	: ARRAY[1..77] OF LREAL := [15377.0, -4587.0, 1374.0, -291.0, -1924.0, -174.0, 358.0, 318.0, 367.0, 132.0, 39.0, -4.0, 82.0, -9.0, -75.0, 66.0, 78.0, 20.0, 29.0, 68.0, 0.0, -25.0, 59.0, -3.0, -3.0, 13.0, 11.0, -45.0, -1.0, -5.0, 13.0, -14.0, 26.0, 15.0, 10.0, 19.0, 2.0, -5.0, 14.0, 4.0, 4.0, -1.0, -4.0, -5.0, 12.0, -3.0, -9.0, 4.0, 1.0, 2.0, 1.0, 3.0, -1.0, 7.0, 2.0, 4.0, -2.0, 3.0, -2.0, 5.0, -4.0, -3.0, -2.0, 0.0, -2.0, 1.0, -2.0, 0.0, -139.0, -2.0, 4.0, 0.0, 0.0, 4.0, -2.0, 2.0, 0.0];

END_VAR

(*
based on:
SOFA Library Issue 2023-10-11 for Fortran 77, nut00b.f

which implements:
 McCarthy, D. and Luzum, B. (2003). "An Abridged Model of
        the Precession & Nutation of the Celestial Pole," Celestial
        Mechanics and Dynamical Astronomy, Volume 85, Issue 1,
        Jan. 2003, p. 37. (IAU 2000B)
NOTES:
- does not implement precession biases (McCarthy, 2003) 2.1
- does implement frame bias offsets as opposed to the SOFA code

IAU 2000B reproduces the IAU 2000A model to a precision
of 1 milliarcsecond in the interval 1995-2050
*)

// Julian centuries FROM J2000 OF jd.
t := (jd -jd2000)/36525.0;

// mean anomaly of the Moon
m_l := LMOD(485868.249036 + t * 1717915923.2178, asec360) * asec2r;

// mean anomaly of the Sun
m_l_ := LMOD(1287104.79305 + t * 129596581.0481, asec360) * asec2r;

// mean argument of the latitude of the Moon
m_f := LMOD(335779.526232 +t * 1739527262.8478, asec360) * asec2r;

// mean elongation of the Moon from the Sun
m_d  := LMOD(1072260.70369 + t * 1602961601.2090, asec360) * asec2r;

// mean longitude of the ascending node of the Moon
m_om  := LMOD(450160.398036 - t * 6962890.5431, asec360) * asec2r;
d_p := 0.0;
d_e := 0.0;
FOR i:=1 TO n_terms BY 1 DO
	theta := LMOD( l[i]*m_l + l_[i]*m_l_ + f[i]*m_f + d[i]*m_d + om[i]*m_om, 2*PI);
	s_theta := SIN(theta);
	c_theta := COS(theta);
	
	d_p := d_p + ((A[i] + A1[i]*t)*s_theta + A2[i]*c_theta);
	d_e := d_e + ((B[i] + B1[i]*t)*c_theta + B2[i]*s_theta);
END_FOR;
// convert from 1e-7 arcsec to arcsec and add planetary nutation terms and frame bias
d_psi := d_p * 1.0E-7 - 0.0433585;
d_eps := d_e * 1.0E-7 - 0.0084531;

END_FUNCTION_BLOCK

// ---- POUs/FUNCTION_BLOCKS/FB_CO_REFRACT.TcPOU
FUNCTION_BLOCK FB_CO_REFRACT
VAR_INPUT
	old_alt			: LREAL;			// old alt in degrees
	altitude		: LREAL := 0.0;		// altitude of observatory
	pressure		: LREAL := 0.0;		// pressure
	temperature		: LREAL := 0.0;		// ground temperature in degrees Celsius, only used if temperature_set is TRUE
	temperature_set	: BOOL := FALSE;	// TRUE: use temperature (0.0 C is valid), FALSE: estimate it from altitude
	epsilon			: LREAL := 0.25; 	//accuracy of iteration for observed=TRUE case, in arcseconds, values below min_epsilon are raised to min_epsilon
	TO_OBSERVED		: BOOL;
END_VAR
VAR_OUTPUT
	new_alt			: LREAL;
	clamped			: BOOL;			// TRUE if altitude, pressure or temperature was outside the model's valid range and has been limited, or old_alt was rejected
END_VAR
VAR
	aout, P, T, dr, cur, last : LREAL;	// P in millibars, T in degrees Celsius
	eps				: LREAL;			// epsilon after clamping
	n				: INT;				// iterations of the observed=TRUE loop
	c				: BOOL;				// clamped flag of one co_refract_forward call
END_VAR
VAR CONSTANT
	alpha 			: LREAL := 0.0065; 	//temp lapse rate [deg C per meter]
	min_epsilon		: LREAL := 0.001;	//smallest accepted epsilon [arcsec]
	max_iterations	: INT := 10;		//iteration cap, the loop converges in 1 to 5 iterations
	max_abs_alt		: LREAL := 1.0E6;	//old_alt beyond this (or NaN/Inf) is rejected
END_VAR

// https://github.com/wlandsman/IDLAstro/blob/master/pro/co_refract.pro

clamped := FALSE;

// Reject NaN/Inf (the comparisons are FALSE for NaN) and pass old_alt through unchanged,
// otherwise the iteration below could not converge.
IF NOT (old_alt > -max_abs_alt AND old_alt < max_abs_alt) THEN
	new_alt := old_alt;
	clamped := TRUE;
	RETURN;
END_IF

// The IDL original works in Kelvin, CO_REFRACT_FORWARD expects degrees Celsius,
// so all temperatures here are Celsius (IDL's 283.0 K and 211.5 K minus the 273.0 offset used there).
IF temperature_set THEN
	T := temperature;
ELSIF altitude > 11000.0 THEN 
	T := 211.5 - 273.0; 
ELSE 
	T := 283.0 - 273.0 - alpha*altitude;
END_IF

// estimate Pressure based on altitude, using U.S. Standard Atmosphere formula.
IF pressure = 0 THEN 
	P := 1010.0*EXPT(1-6.5/288000*altitude, 5.255);
ELSE
	P := pressure;
END_IF

IF NOT TO_OBSERVED THEN 
	aout := old_alt - co_refract_forward(old_alt, P:=P, T:=T, clamped => c);
	clamped := c;
ELSE
	aout := 0.0;
	//calculate initial refraction guess
	dr := co_refract_forward(old_alt, P:=P, T:=T, clamped => c);
	clamped := c;
	cur := old_alt + dr; // guess of observed location

	// epsilon <= 0 (or NaN) would never satisfy the exit condition, so clamp it and cap the iterations
	IF epsilon > min_epsilon THEN
		eps := epsilon;
	ELSE
		eps := min_epsilon;
	END_IF
	n := 0;
	REPEAT 
	 	last := cur;
		dr := co_refract_forward(cur, P:= P, T:=T, clamped => c);
		clamped := clamped OR c;
	  	cur := old_alt + dr;
		n := n + 1;
	UNTIL ABS(last-cur)*3600.0 < eps OR n >= max_iterations
	END_REPEAT
	aout := cur;
END_IF

new_alt := aout;

END_FUNCTION_BLOCK

// ---- POUs/FUNCTION_BLOCKS/FB_CO_NUTATE.TcPOU
FUNCTION_BLOCK FB_CO_NUTATE
VAR_INPUT
	jd			: LREAL;		// Julian date
	ra			: LREAL;		// RA in degrees
	dec			: LREAL;		// Dec in degrees
	nut_given	: BOOL := FALSE;	// TRUE: d_psi_in/d_eps_in already hold the nutation of jd, it is not evaluated again
	d_psi_in	: LREAL;		// nutation in longitude in arcsec (only used if nut_given)
	d_eps_in	: LREAL;		// nutation in obliquity in arcsec (only used if nut_given)
END_VAR
VAR_OUTPUT
	d_ra		: LREAL;		// RA diff in degrees
	d_dec		: LREAL;		// Dec diff in degrees
	eps			: LREAL;		// TRUE obliquity OF the ecliptic in radians
	d_psi		: LREAL;		// in arcsec
	d_eps		: LREAL;
END_VAR
VAR
	ce, se,x,y,z,x2,y2,z2,rad,xyproj,ra2,dec2: LREAL;
	nutate		: FB_IAU2000B;
END_VAR
VAR CONSTANT
	d2r			: LREAL := PI/180.0;
	d2as		: LREAL := PI/(180.0*3600.0);
END_VAR

// https://github.com/wlandsman/IDLAstro/blob/master/pro/co_nutate.pro
(*EXPLANATION:
;     Calculates necessary changes to ra and dec due to
;     the nutation of the Earth's rotation axis, as described in Meeus, Chap 23.
;     Uses formulae from Astronomical Almanac, 1984, and does the calculations
;     in equatorial rectangular coordinates to avoid singularities at the
;     celestial poles.*)
// must calculate obliquity OF ecliptic
IF nut_given THEN
	d_psi := d_psi_in;
	d_eps := d_eps_in;
ELSE
	nutate(jd := jd,
			d_psi => d_psi,
			d_eps => d_eps);
END_IF

eps := JD2OBLIQUITY(jd, d_eps); // TRUE obliquity OF the ecliptic in radians
 
//useful numbers
ce := COS(eps);
se := SIN(eps);

// convert ra-dec to equatorial rectangular coordinates
x := COS(ra*d2r) * COS(dec*d2r);
y := SIN(ra*d2r) * COS(dec*d2r);
z := SIN(dec*d2r);

// apply corrections to each rectangular coordinate
x2 := x - (y*ce + z*se)*d_psi * d2as;
y2 := y + (x*ce*d_psi - z*d_eps) * d2as;
z2 := z + (x*se*d_psi + y*d_eps) * d2as;

// convert back to equatorial spherical coordinates
rad := SQRT(x2*x2 + y2*y2 + z2*z2);
xyproj := SQRT(x2*x2 + y2*y2);

ra2  := x2 * 0.0;
dec2 := x2 * 0.0;

// Calculate Ra and Dec in RADIANS (later convert to DEGREES)
IF (xyproj = 0) AND (z <> 0) THEN
	// places where xyproj=0 (point at NCP or SCP)
	dec2 := ASIN(LIMIT(-1.0, z2/rad, 1.0));
	ra2 := 0.0;
END_IF
 
IF (xyproj <> 0) THEN
	// places other than NCP or SCP
	ra2 := ATAN2(y2, x2);
	dec2 := ASIN(LIMIT(-1.0, z2/rad, 1.0));
END_IF

// convert to DEGREES

ra2 := ra2 /d2r;
dec2 := dec2 /d2r;

ra2 := MODABS(ra2, 360.0);


// Return changes in ra and dec
// wrap to +-180 so that an unwrapped input ra (e.g. -5) or ra2 across 0/360 gives a small difference
d_ra := MODABS(ra2 - ra + 180.0, 360.0) - 180.0;
d_dec := (dec2 - dec);

END_FUNCTION_BLOCK

// ---- POUs/FUNCTION_BLOCKS/FB_EQ2HOR.TcPOU
FUNCTION_BLOCK FB_EQ2HOR
VAR_INPUT
	ra				: LREAL;	// right ascension in degrees
	dec				: LREAL;	// declination in degrees
	jd				: LREAL;	// Julian Date, UTC time scale
	dut1			: LREAL := 0.0;	// UT1-UTC in seconds (IERS), 0 treats UTC as UT1
	lon				: LREAL;	// longitude in degrees
	lat				: LREAL;	// latitude in degrees
	ws				: BOOL := FALSE; 	// Set this to TRUE get the azimuth measured westward FROM south (NOT East of North).
	precess			: BOOL := TRUE; 	// Set this to 1 to force precession [default], 0 for no precession correction
	nutate			: BOOL := TRUE; 	// Set this to 1 to force nutation [default], 0 for no nutation correction.
	aberration		: BOOL := TRUE; 	// Set this to 1 to force aberration correction [default], 0 for no correction.
	refract 		: BOOL := TRUE; 	// Set to 1 to force refraction correction[default] (for actual sky coord), 0 for no correction (for theoretical coord).
	refract_to_observed : BOOL := TRUE;
	altitude		: LREAL := 0.0;
END_VAR
VAR_OUTPUT
	alt				: LREAL;		// altitude in degrees
	az				: LREAL;		// azimuth in degrees
	ha				: LREAL;		// hour angle in degrees
END_VAR
VAR
	radec2hadec		: FB_RADEC2HADEC;
	hadec2altaz		: FB_HADEC2ALTAZ;
	co_refract		: FB_CO_REFRACT;
	dec_app			: LREAL;		// Apparent Dec in degrees
END_VAR

(* source https://github.com/wlandsman/IDLAstro/blob/master/pro/eq2hor.pro 

PURPOSE:
	Convert celestial  (ra-dec) coords to local horizon coords (alt-az).

DESCRIPTION:
This  code calculates horizon (alt,az) coordinates from equatorial
(ra,dec) coords. It is typically accurate to about 1 arcsecond or better (I
have checked the output against the publicly available XEPHEM software). It
performs precession, nutation, aberration, and refraction corrections. [...]
*)


// precession, nutation and aberration (each one optional), then the hour angle
radec2hadec(
	jd := jd,
	dut1 := dut1,
	ra := ra,
	dec := dec,
	lon := lon,
	precess := precess,
	nutate := nutate,
	aberration := aberration,
	ha_out => ha,
	dec_out => dec_app);

(*******************************************************************************
 Now do the spherical trig to get APPARENT alt,az. *)
hadec2altaz(	
	ha := ha, 
	dec := dec_app, 
	lat := lat, 
	alt => alt, 
	az => az, 
	WS := WS);

(********************************************************************************************
 Make Correction for ATMOSPHERIC REFRACTION
 (use this for visible and radio wavelengths; author is unsure about other wavelengths.
  See the comments in CO_REFRACT for more details.) *)
IF refract THEN 
	co_refract(	
		old_alt := alt, 
		altitude := altitude, 
		to_observed := refract_to_observed, 
		new_alt => alt);
END_IF

END_FUNCTION_BLOCK

// ---- POUs/FUNCTION_BLOCKS/FB_RADEC2HADEC.TcPOU
FUNCTION_BLOCK FB_RADEC2HADEC
VAR_INPUT
	jd				: LREAL;		// Julian date, UTC time scale
	dut1			: LREAL := 0.0;	// UT1-UTC in seconds (IERS), 0 treats UTC as UT1
	ra				: LREAL;		// Right Ascension (ICRS) in degrees
	dec				: LREAL;		// Declination (ICRS) in degrees
	lon				: LREAL;		// Longitude in degrees
	precess			: BOOL := TRUE;	// FALSE: no precession correction
	nutate			: BOOL := TRUE;	// FALSE: no nutation correction
	aberration		: BOOL := TRUE;	// FALSE: no aberration correction
END_VAR
VAR_OUTPUT
	ha_out			: LREAL;		// Hour angle (APPARENT) in degrees
	dec_out			: LREAL;		// Declination (APPARENT) in degrees
END_VAR
VAR
	lmst			: LREAL;
	last			: LREAL;
	d_psi			: LREAL;
	d_eps			: LREAL;
	eps				: LREAL;
	J_now			: LREAL;
	IAU2000B		: FB_IAU2000B;
	fbprecess		: FB_PRECESS;
	co_nutate		: FB_CO_NUTATE;
	co_aberration	: FB_CO_ABERRATION;
	d_ra_abr		: LREAL;		// Difference in RA due to aberration
	d_dec_abr		: LREAL;		// Difference in Dec due to aberration
	d_ra_nut		: LREAL;		// Difference in RA due to nutation
	d_dec_nut		: LREAL;		// Difference in Dec due to nutation
	ra_pre, dec_pre	: LREAL;		// precessed coords
	ra_app, dec_app	: LREAL;		// apparent coords
END_VAR

// This code calculates the Hour Angle and Declination (APPARENT) from the Right Ascension and Declination (ICRS)
// This includes P03 precession and IAU2000B nutation as well as aberration (IDL libary)
// adapted from: https://github.com/wlandsman/IDLAstro/blob/master/pro/eq2hor.pro (IDL libary)
// this version is written by Lukas Melzig
// the corrections are only written below if the respective flag is set, so start from zero
// to not keep applying the values of a previous call
d_ra_nut := 0.0;
d_dec_nut := 0.0;
d_ra_abr := 0.0;
d_dec_abr := 0.0;

(* ******************************************************************************
 PRECESS coordinates to current date
 (uses astro lib procedure PRECESS.pro)
*)
J_now := JD2JEPOCH(jd); // compute current equinox
IF precess THEN
	fbprecess(
		ra := ra,
		dec := dec,
		equinox1 := 2000.0,
		equinox2 := J_now,
		ra_precessed => ra_pre,
		dec_precessed => dec_pre);
ELSE
	ra_pre := ra;
	dec_pre := dec;
END_IF

(******************************************************************************
 calculate NUTATION and ABERRATION Corrections to Ra-Dec
*)

// d_psi and eps are also needed for the sidereal time if nutation is not applied
IAU2000B(jd := jd,
		d_psi => d_psi,
		d_eps => d_eps);
eps := JD2OBLIQUITY(jd, d_eps); // TRUE obliquity OF the ecliptic in radians

IF nutate THEN
	co_nutate(
		jd := jd,
		ra := ra_pre,
		dec := dec_pre,
		nut_given := TRUE,
		d_psi_in := d_psi,
		d_eps_in := d_eps,
		d_ra => d_ra_nut,
		d_dec => d_dec_nut);
END_IF

IF aberration THEN
	co_aberration(
		jd := jd,
		ra := ra_pre,
		dec := dec_pre,
		d_ra => d_ra_abr,
		d_dec => d_dec_abr,
		eps := eps);
END_IF
ra_app := ra_pre + d_ra_abr + d_ra_nut;
dec_app := dec_pre + d_dec_abr + d_dec_nut;
(***************************************************************************************
Calculate LOCAL MEAN SIDEREAL TIME *)
lmst := jd2lst(JD:=jd, lon:=lon, dut1:=dut1);
// calculate local APPARENT sidereal time
last := LMST2LAST(lmst, d_psi, eps);

(******************************************************************************
 Find hour angle (in DEGREES) *)
ha_out := last - ra_app;
ha_out := MODABS(ha_out, 360.0);
// apparent declination
dec_out := dec_app;

END_FUNCTION_BLOCK

// ---- POUs/FUNCTION_BLOCKS/FB_PRECESS.TcPOU
FUNCTION_BLOCK FB_PRECESS
VAR_INPUT
	ra				: LREAL;		// RA in degrees
	dec				: LREAL;		// Dec in degrees
	equinox1		: LREAL;		// epoch (Julian year) of the input coordinates
	equinox2		: LREAL;		// epoch (Julian year) of the output coordinates
END_VAR
VAR_OUTPUT
	ra_precessed	: LREAL;
	dec_precessed	: LREAL;
END_VAR
VAR
	ra_rad			: LREAL;		// RA in rad
	dec_rad			: LREAL;		// Dec in rad
	t				: LREAL;		// the elapsed time in Julian centuries since J2000 TT (days)
	EPS0, PSIA, OMEGAA, CHIA : LREAL;
	x, x2			: ARRAY[0..2] OF LREAL;
	rot				: ARRAY[0..2,0..2] OF LREAL;
	SA, CA, SB,CB,SC,CC,SD,CD: LREAL;
	step			: INT;			// 0: equinox1 -> J2000, 1: J2000 -> equinox2
	epoch			: LREAL;		// the non-J2000 epoch of the current step
END_VAR
VAR CONSTANT
	d2r 			: LREAL := PI/180.0;
	sec_to_rad 		: LREAL := d2r/3600.0;
END_VAR

(*
based on: NOVAS_F3.1.f -> SUBROUTINE PRECES
Kaplan, G., Bartlett, J., Monet, A., Bangert, J., & Puatua, W. (2011) User's Guide to NOVAS Version F3.1 (Washington, DC: USNO).

 THIS SUBROUTINE PRECESSES EQUATORIAL RECTANGULAR COORDINATES FROM
 ONE EPOCH TO ANOTHER.  THE COORDINATES ARE REFERRED TO THE MEAN
 DYNAMICAL EQUATOR AND EQUINOX OF THE TWO RESPECTIVE EPOCHS.  SEE
 EXPLANATORY SUPPLEMENT TO THE ASTRONOMICAL ALMANAC, PP. 103-104,
 AND CAPITAINE ET AL. (2003), ASTRONOMY AND ASTROPHYSICS 412,
 567-586.

 PRECES only rotates between J2000 and one other epoch, so a general
 equinox1 -> equinox2 is done in two steps via J2000. A step whose epoch
 is exactly 2000.0 is the identity and skipped.
*)

// deg 2 radian
ra_rad := ra*d2r;
dec_rad := dec*d2r;

x[0] := COS(dec_rad )*COS(ra_rad);
x[1] := COS(dec_rad )*SIN(ra_rad);
x[2] := SIN(dec_rad);


IF equinox1 <> equinox2 THEN
	FOR step := 0 TO 1 DO
		IF step = 0 THEN
			epoch := equinox1;
		ELSE
			epoch := equinox2;
		END_IF
		IF epoch <> 2000.0 THEN
			// t is the elapsed time in Julian centuries between J2000 and epoch
			t := 0.01*(epoch - 2000.0);
			EPS0 := sec_to_rad*	84381.406;
			PSIA := sec_to_rad*	( ( ( ( -    0.0000000951   * t
										+    0.000132851  ) * t
										-    0.00114045   ) * t
										-    1.0790069    ) * t
										+ 5038.481507     ) * t;
			OMEGAA := sec_to_rad*	( ( ( ( +    0.0000003337   * t
											-    0.000000467  ) * t
											-    0.00772503   ) * t
											+    0.0512623    ) * t
											-    0.025754     ) * t + EPS0;
			CHIA   := sec_to_rad*	( ( ( ( -    0.0000000560   * t
											+    0.000170663  ) * t
											-    0.00121197   ) * t
											-    2.3814292    ) * t
											+   10.556403     ) * t;
			SA := SIN(EPS0);
			CA := COS( EPS0 );
			SB := SIN( -PSIA );
			CB := COS( -PSIA );
			SC := SIN( -OMEGAA );
			CC := COS( -OMEGAA );
			SD := SIN( CHIA );
			CD := COS( CHIA );

			// COMPUTE ELEMENTS OF PRECESSION ROTATION MATRIX
			// EQUIVALENT TO R3(CHI_A)R1(-OMEGA_A)R3(-PSI_A)R1(EPSILON_0)
			rot[0,0] :=  CD * CB - SB * SD * CC; 	rot[0,1] := CD * SB * CA + SD * CC * CB * CA - SA * SD * SC; 	rot[0,2] := CD * SB * SA + SD * CC * CB * SA + CA * SD * SC;
			rot[1,0] := -SD * CB - SB * CD * CC; 	rot[1,1] := -SD * SB * CA + CD * CC * CB * CA - SA * CD * SC; 	rot[1,2] := -SD * SB * SA + CD * CC * CB * SA + CA * CD * SC;
			rot[2,0] := SB * SC;					rot[2,1] := -SC * CB * CA - SA * CC; 							rot[2,2] := -SC * CB * SA + CC * CA;

			// calculation as: Explanatory Supplement to the Astronomical Almanac (2013) p.220 eq.6.30
			//x2 := rot* x; //rotate to get output direction cosines
			IF step = 0 THEN
				// PERFORM ROTATION FROM EPOCH (equinox1) TO J2000.0
				x2[0] := rot[0,0]*x[0] + rot[1,0]*x[1] + rot[2,0]*x[2];
				x2[1] := rot[0,1]*x[0] + rot[1,1]*x[1] + rot[2,1]*x[2];
				x2[2] := rot[0,2]*x[0] + rot[1,2]*x[1] + rot[2,2]*x[2];
			ELSE
				// PERFORM ROTATION FROM J2000.0 TO EPOCH (equinox2)
				x2[0] := rot[0,0]*x[0] + rot[0,1]*x[1] + rot[0,2]*x[2];
				x2[1] := rot[1,0]*x[0] + rot[1,1]*x[1] + rot[1,2]*x[2];
				x2[2] := rot[2,0]*x[0] + rot[2,1]*x[1] + rot[2,2]*x[2];
			END_IF
			x[0] := x2[0];
			x[1] := x2[1];
			x[2] := x2[2];
		END_IF
	END_FOR
END_IF


ra_rad := atan2(x[1],x[0]);
dec_rad := ASIN(LIMIT(-1.0, x[2], 1.0));

ra_precessed := ra_rad/d2r;
ra_precessed := MODABS(ra_precessed, 360.0);            //RA between 0 AND 360 degrees
dec_precessed := dec_rad/d2r;

END_FUNCTION_BLOCK

// ---- POUs/FUNCTION_BLOCKS/FB_HADEC2ALTAZ.TcPOU
FUNCTION_BLOCK FB_HADEC2ALTAZ
VAR_INPUT
	ha				: LREAL;		// Hour angle in degrees
	dec				: LREAL;		// Declination in degrees
	lat				: LREAL;		// Latitude in degrees
	WS				: BOOL := FALSE;
END_VAR
VAR_OUTPUT
	alt				: LREAL;		// altitude in degrees
	az				: LREAL;		// azimuth in degrees
END_VAR
VAR
	sh,sd,sl, ch,cd,cl,	x, y, z, radius: LREAL;
END_VAR
VAR CONSTANT
	d2r 			: LREAL := PI/180.0;
END_VAR

(* source https://github.com/wlandsman/IDLAstro/blob/master/pro/hadec2altaz.pro
;+
;  NAME:
;     HADEC2ALTAZ
;  PURPOSE:
;      Converts Hour Angle and Declination to Horizon (alt-az) coordinates.
;  EXPLANATION:
;      Can deal with NCP/SCP singularity.    Intended mainly to be used by
;      program EQ2HOR
;
; CALLING SEQUENCE:
;      HADEC2ALTAZ, ha, dec, lat ,alt ,az [ /WS ]
;
; INPUTS
;     ha -  the local apparent hour angle, in DEGREES, scalar or vector
;     dec -  the local apparent declination, in DEGREES, scalar or vector
;     lat -  the local latitude, in DEGREES, scalar or vector
;
; OUTPUTS
;     alt - the local apparent altitude, in DEGREES.
;     az  - the local apparent azimuth, in DEGREES, all results in double
;           precision
; OPTIONAL KEYWORD INPUT:
;      /WS - Set this keyword for the output azimuth to be measured West from 
;            South.    The default is to measure azimuth East from North.
;
; EXAMPLE:
;     What were the apparent altitude and azimuth of the sun when it transited 
;     the local meridian at Pine Bluff Observatory (Lat=+43.07833 degrees) on 
;     April 21, 2002?   An object transits the local meridian at 0 hour angle.
;     Assume this will happen at roughly 1 PM local time (18:00 UTC).
;
;     IDL> jdcnv, 2002, 4, 21, 18., jd  ; get rough Julian date to determine 
;                                       ;Sun ra, dec.
;     IDL> sunpos, jd, ra, dec
;     IDL> hadec2altaz, 0., dec, 43.078333, alt, az
;
;       ===> Altitude alt = 58.90
;            Azimuth  az = 180.0

; REVISION HISTORY:
;      Written  Chris O'Dell Univ. of Wisconsin-Madison May 2002
;-
*)
sh := SIN(ha*d2r);
ch := COS(ha*d2r);
sd := SIN(dec*d2r);
cd := COS(dec*d2r);
sl := SIN(lat*d2r);
cl := COS(lat*d2r);

x := -ch * cd * sl + sd * cl;
y := -sh * cd;
z := ch * cd * cl + sd * sl;
radius := SQRT(x*x + y*y);

// now get Alt, Az
az := ATAN2(y, x) /d2r;	// was ATAN(y, x)
alt := ATAN2(z, radius) / d2r;

// correct for negative AZ
az := MODABS(az, 360.0);

// convert AZ to West from South, if desired
IF WS THEN 
	az := MODABS(az + 180.0, 360);
END_IF

END_FUNCTION_BLOCK

// ---- POUs/FUNCTION_BLOCKS/FB_HADEC2RADEC.TcPOU
FUNCTION_BLOCK FB_HADEC2RADEC
VAR_INPUT
	jd				: LREAL;		// Julian date, UTC time scale
	dut1			: LREAL := 0.0;	// UT1-UTC in seconds (IERS), 0 treats UTC as UT1
	ha				: LREAL;		// Hour angle (APPARENT) in degrees
	dec				: LREAL;		// Declination (APPARENT) in degrees
	lon				: LREAL;		// Longitude in degrees
	precess			: BOOL := TRUE;	// FALSE: no precession correction
	nutate			: BOOL := TRUE;	// FALSE: no nutation correction
	aberration		: BOOL := TRUE;	// FALSE: no aberration correction
END_VAR
VAR_OUTPUT
	ra_out				: LREAL;		// RA in degrees (ICRS)
	dec_out			: LREAL;			// DEC in degrees (ICRS)
END_VAR
VAR
	lmst			: LREAL;
	last			: LREAL;
	d_psi			: LREAL;
	d_eps			: LREAL;
	eps				: LREAL;
	J_now			: LREAL;
	IAU2000B		: FB_IAU2000B;
	fbprecess		: FB_PRECESS;
	co_nutate		: FB_CO_NUTATE;
	co_aberration	: FB_CO_ABERRATION;
	d_ra_abr		: LREAL;		// Difference in RA due to aberration
	d_dec_abr		: LREAL;		// Difference in Dec due to aberration
	d_ra_nut		: LREAL;		// Difference in RA due to nutation
	d_dec_nut		: LREAL;		// Difference in Dec due to nutation
	alt,az			: LREAL;
END_VAR

// This code calculates the Right Ascension and Declination (ICRS) from the Hour Angle and Declination (APPARENT)
// This includes P03 precession and IAU2000B nutation as well as aberration (IDL libary)
// adapted from: https://github.com/wlandsman/IDLAstro/blob/master/pro/hor2eq.pro (IDL libary)
// this version is written by Lukas Melzig


// the corrections are only written below if the respective flag is set, so start from zero
// to not keep applying the values of a previous call
d_ra_nut := 0.0;
d_dec_nut := 0.0;
d_ra_abr := 0.0;
d_dec_abr := 0.0;

// must calculate obliquity OF ecliptic
IAU2000B(jd := jd,
		d_psi => d_psi,
		d_eps => d_eps);

eps := JD2OBLIQUITY(jd, d_eps); // TRUE obliquity OF the ecliptic in radians

// Calculate LOCAL MEAN SIDEREAL TIME
lmst := jd2lst(JD:=jd, lon:=lon, dut1:=dut1);
// calculate local APPARENT sidereal time
last := LMST2LAST(lmst, d_psi, eps);

// Find right ascension (in DEGREES)
ra_out := MODABS(last - ha + 360.0, 360.0);
dec_out := dec;
//*****************************************************************************
// calculate NUTATION and ABERRATION Corrections to Ra-Dec
IF nutate THEN
	co_nutate(
		jd := jd,
		ra := ra_out,
		dec := dec_out,
		nut_given := TRUE,
		d_psi_in := d_psi,
		d_eps_in := d_eps,
		d_ra => d_ra_nut,
		d_dec => d_dec_nut);
END_IF

IF aberration THEN
	co_aberration(
		jd := jd,
		ra := ra_out,
		dec := dec_out,
		eps := eps,
		d_ra => d_ra_abr,
		d_dec => d_dec_abr);
END_IF
//apply
ra_out := ra_out - (d_ra_abr + d_ra_nut);
dec_out := dec_out - (d_dec_abr + d_dec_nut);
//*****************************************************************************
//precess back
J_now := JD2JEPOCH(jd); // compute current equinox
IF precess THEN
	fbprecess(
		ra := ra_out,
		dec := dec_out,
		equinox1 := J_now,
		equinox2 := 2000.0,
		ra_precessed => ra_out,
		dec_precessed => dec_out);
ELSE
	// the precession block wraps RA, without it the correction can leave 0 to 360
	ra_out := MODABS(ra_out, 360.0);
END_IF

END_FUNCTION_BLOCK

// ---- POUs/FUNCTION_BLOCKS/FB_HOR2EQ.TcPOU
FUNCTION_BLOCK FB_HOR2EQ
VAR_INPUT
	alt				: LREAL;			//altitude (in degrees)  
	az				: LREAL;			//azimuth angle (in degrees, measured EAST from NORTH, but see keyword WS below.) [scalar or vector]
	jd				: LREAL;			// Julian Date, UTC time scale
	dut1			: LREAL := 0.0;	// UT1-UTC in seconds (IERS), 0 treats UTC as UT1
	lat				: LREAL;			// observers latitude (degrees)
	lon				: LREAL;			// observers longitude (degrees)
	ws				: BOOL := FALSE; 	// Set this to TRUE get the azimuth measured westward FROM south (NOT East of North).
	precess			: BOOL := TRUE; 	// Set this to 1 to force precession [default], 0 for no precession correction
	nutate			: BOOL := TRUE; 	// Set this to 1 to force nutation [default], 0 for no nutation correction.
	aberration		: BOOL := TRUE; 	// Set this to 1 to force aberration correction [default], 0 for no correction.
	refract			: BOOL := TRUE; 	// Set to 1 to force refraction correction[default] (for actual sky coord), 0 for no correction (for theoretical coord).
	altitude		: LREAL := 0.0;
	alt_is_observed	: BOOL := TRUE;		// TRUE: alt is an observed (refracted) altitude, refraction is removed [default]. FALSE: alt is geometric, refraction is added. Only used if refract is TRUE.
END_VAR
VAR_OUTPUT
	ra				: LREAL;			// Right Ascension of object  (J2000) in degrees (FK5)
	dec				: LREAL;			// Declination of object (J2000) in degrees (FK5)
	ha				: LREAL;			// hour angle (in degrees) (optional)
END_VAR
VAR
	co_refract		: FB_CO_REFRACT;
	altaz2hadec		: FB_ALTAZ2HADEC;
	hadec2radec		: FB_HADEC2RADEC;
	d_dec_ref		: LREAL;		// time reference
	alt_loc			: LREAL;		// altitude after refraction correction
	az_loc			: LREAL;		// azimuth measured east from north

END_VAR
VAR CONSTANT
	// easier then functions
	h2d				: LREAL := 15.0;
END_VAR

(* https://github.com/wlandsman/IDLAstro/blob/master/pro/hor2eq.pro
; NAME:
;   HOR2EQ
;
; PURPOSE:
;    Converts local horizon coords (alt-az) of something to equatorial (ra-dec).
;
; EXPLANATION:
;     This is a nice code to calculate equatorial (ra,dec) coordinates from
;     horizon (alt,az) coords.    It is typically accurate to about 1 arcsecond
;     or better (I have checked the output against the publicly available XEPHEM
;     software). It performs precession, nutation, aberration, and refraction
;     corrections.  The perhaps best thing about it is that it can take arrays
;     as inputs, in all variables and keywords EXCEPT Lat, lon, and Altitude
;    (the code assumes these aren't changing), and uses vector arithmetic in
;     every calculation except when calculating the precession matrices.
;
; DEPENDENCIES:
;       NUTATE, PRECESS, SUNPOS,
;       CO_NUTATE, CO_ABERRATION, CO_REFRACT, HADEC2ALTAZ
;CORRECTIONS I DO NOT MAKE:
;   *  Deflection of Light by the sun due to GR. (typically milliarcseconds,
;        can be arcseconds within one degree of the sun)
;   *  The Effect of Annual Parallax (typically < 1 arcsecond)
;   *  and more (see below)
;
; TO DO
;    * Better Refraction Correction.  Need to put in wavelength dependence,
;       and integrate through the atmosphere.
;    * Topocentric Parallax Correction (will take into account elevation of
;          the observatory)
;    * Proper Motion (but this will require crazy lookup tables or something).
;    * Difference between UTC and UT1 in determining LAST -- is this important?
;    * Effect of Annual Parallax (is this the same as topocentric Parallax?)
;    * Polar Motion
;    * Better connection to Julian Date Calculator.
;
; AUTHOR:
;   Chris O'Dell
;   Assistant Professor of Atmospheric Science
;   Colorado State University
;   Email: odell@atmos.colostate.edu
; REVISION HISTORY:
;     Made all integers type LONG  W. Landsman   September 2007
;     Fixed for case of scalar Julian date but vector positions W L June 2009
;-*)

az_loc := az;
IF WS THEN 
	az_loc := az - 180.0;
END_IF

(********************************************************************************************
 Make Correction for ATMOSPHERIC REFRACTION
 (use this for visible and radio wavelengths; author is unsure about other wavelengths.
  See the comments in CO_REFRACT for more details.) *)
alt_loc := alt;
IF refract THEN 
	co_refract(	
		old_alt := alt, 
		altitude := altitude, 
		to_observed := NOT alt_is_observed, 
		new_alt => alt_loc);
END_IF


//****************************************************************************
// Now do the spherical trig to get APPARENT Hour Angle [degrees], and
// declination [degrees].
altaz2hadec(alt := alt_loc, az := az_loc, lat := lat, ha => ha, dec => dec);

//*****************************************************************************
// Right Ascension (in degrees, from 0 to 360.): local apparent sidereal time, then
// the corrections for nutation, aberration and precession back to J2000
hadec2radec(
	jd := jd,
	dut1 := dut1,
	ha := ha,
	dec := dec,
	lon := lon,
	precess := precess,
	nutate := nutate,
	aberration := aberration,
	ra_out => ra,
	dec_out => dec);

END_FUNCTION_BLOCK
